(* Schneider Machine Expert - Basic project Tank_Level_Control, file version 3.0.0.0 *)
(* ProjectInformations: Name=Tank_Level_Control *)

HARDWARE
  Cpu 0: TM221CE16T
  Extension 0: TM3AI4
  EthernetConfiguration: NetworkName=M221, IpAllocationMode=ByDhcp, IpAddress=192.168.1.10, SubnetMask=255.255.255.0
  SerialLineConfiguration: Baud=Baud19200, Parity=ParityEven, DataBits=DataBits8, StopBits=StopBits1, PhysicalMedium=PhysicalMediumRs485, TransmissionMode=TransmissionModeModbusRtu, SlaveId=1, Addressing=SlaveAddressing
  MastTask: UsePeriodScanMode=false, PeriodScan=100
  FastTask: Period=255
  CpuBehavior: StartingMode=StartAsPreviousState, AutoSaveRamOnEeprom=true, WatchdogPeriod=250

SYMBOLS  (address, symbol, comment, settings)
  %M0       TANK_FULL  "Tank full flag from ultrasonic"
  %M1       TANK_EMPTY  "Tank empty flag from ultrasonic"
  %Q0.0     INLET_VLV
  %Q0.1     OUTLET_VLV
  %IW1.0    LEVEL_AIN  "Ultrasonic level transmitter 4-20mA"  [AIType=Current4_20mA, AIRange=Range0_10000, AIFilter=AIFilter4]

POU Main Program
  (* SectionNumber=1 *)

// Rung 0: Tank Full Detection
// Set flag when ultrasonic reads low (tank full)
  LD [%IW1.0<1800]        (* LEVEL_AIN *)
  ST %M0                  (* TANK_FULL *)
  // as ST:
  //   TANK_FULL := LEVEL_AIN<1800;
  (* the ladder stored for this rung does not match its IL; not drawn *)

// Rung 1: Tank Empty Detection
// Set flag when ultrasonic reads high (tank empty)
  LD [%IW1.0>4800]        (* LEVEL_AIN *)
  ST %M1                  (* TANK_EMPTY *)
  // as ST:
  //   TANK_EMPTY := LEVEL_AIN>4800;
  (* the ladder stored for this rung does not match its IL; not drawn *)

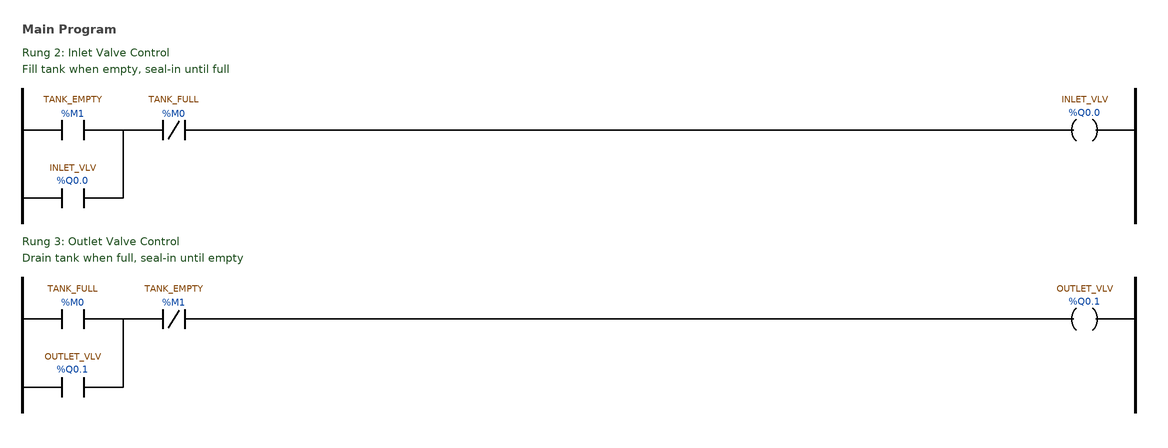

// Rung 2: Inlet Valve Control
// Fill tank when empty, seal-in until full
  LD %M1                  (* TANK_EMPTY *)
  OR %Q0.0                (* INLET_VLV *)
  ANDN %M0                (* TANK_FULL *)
  ST %Q0.0                (* INLET_VLV *)
  // as ST:
  //   INLET_VLV := (TANK_EMPTY OR INLET_VLV) AND NOT TANK_FULL;

// Rung 3: Outlet Valve Control
// Drain tank when full, seal-in until empty
  LD %M0                  (* TANK_FULL *)
  OR %Q0.1                (* OUTLET_VLV *)
  ANDN %M1                (* TANK_EMPTY *)
  ST %Q0.1                (* OUTLET_VLV *)
  // as ST:
  //   OUTLET_VLV := (TANK_FULL OR OUTLET_VLV) AND NOT TANK_EMPTY;
